FUNCTION_BLOCK PAMParkingspace EXTENDS PAProcessModule
VAR_INPUT
END_VAR
VAR_OUTPUT
END_VAR
VAR
	_PAPointMatIn1 : PAPoint(THIS^);
	_PAPointMatOut1 : PAPoint(THIS^);
END_VAR

METHOD FB_init : BOOL
VAR_INPUT
	bInitRetains : BOOL; // if TRUE, the retain variables are initialized (warm start / cold start)
	bInCopyCode : BOOL;  // if TRUE, the instance afterwards gets moved into the copy code (online change)
	parent : IACComponent;
END_VAR
AddPoint(_PAPointMatIn1);
AddPoint(_PAPointMatOut1);
END_METHOD

PROPERTY PUBLIC PAPointMatIn1 : IACPoint
GET
PAPointMatIn1 := _PAPointMatIn1;
END_GET
END_PROPERTY

PROPERTY PUBLIC PAPointMatOut1 : IACPoint
GET
PAPointMatOut1 := _PAPointMatOut1;
END_GET
END_PROPERTY

END_FUNCTION_BLOCK

(* stored: Version 1.1.0.1, ProductVersion 3.1.4020.12
   POU PAMParkingspace: Id {944ded07-cb87-47d9-ad64-4dbcf8e5819e}, SpecialFunc None
   Method FB_init: Id {e96acda6-b8b0-4d96-9028-eef59c0be988}
   Property PAPointMatIn1: Id {ec09795e-bfa8-415e-8217-b137d104c328}
   Get Get: Id {ad917246-eb45-447d-bdce-cb991b5e2c96}
   Property PAPointMatOut1: Id {1c17f1e2-ab65-4f77-a427-18f47edd5d8d}
   Get Get: Id {924a6b4f-9faa-42a8-a1ea-23f02e17aed5} *)
